(* Schneider Machine Expert - Basic project LT, file version 1.7.0.0 *)
(* ProjectInformations: Name=New project *)

HARDWARE
  Cpu 0: TM221ME32TK
  EthernetConfiguration: NetworkName=M221, IpAllocationMode=FixedAddress, IpAddress=0.0.0.0, SubnetMask=0.0.0.0
  SerialLineConfiguration: Baud=Baud19200, Parity=ParityEven, DataBits=DataBits8, StopBits=StopBits1, PhysicalMedium=PhysicalMediumRs485, TransmissionMode=TransmissionModeModbusRtu, SlaveId=1, Addressing=SlaveAddressing
  MastTask: UsePeriodScanMode=false, PeriodScan=100
  FastTask: Period=255
  CpuBehavior: StartingMode=StartAsPreviousState, AutoSaveRamOnEeprom=true, WatchdogPeriod=250

SYMBOLS  (address, symbol, comment, settings)
  %Q0.0       "P1"
  %Q0.1       "P2"
  %Q0.2       "SOV"
  %IW0.0      [Type=Type_0_10V, Scope=Scope_Normal, Minimum=0, Maximum=1000]

POU New POU
  (* SectionNumber=1 *)

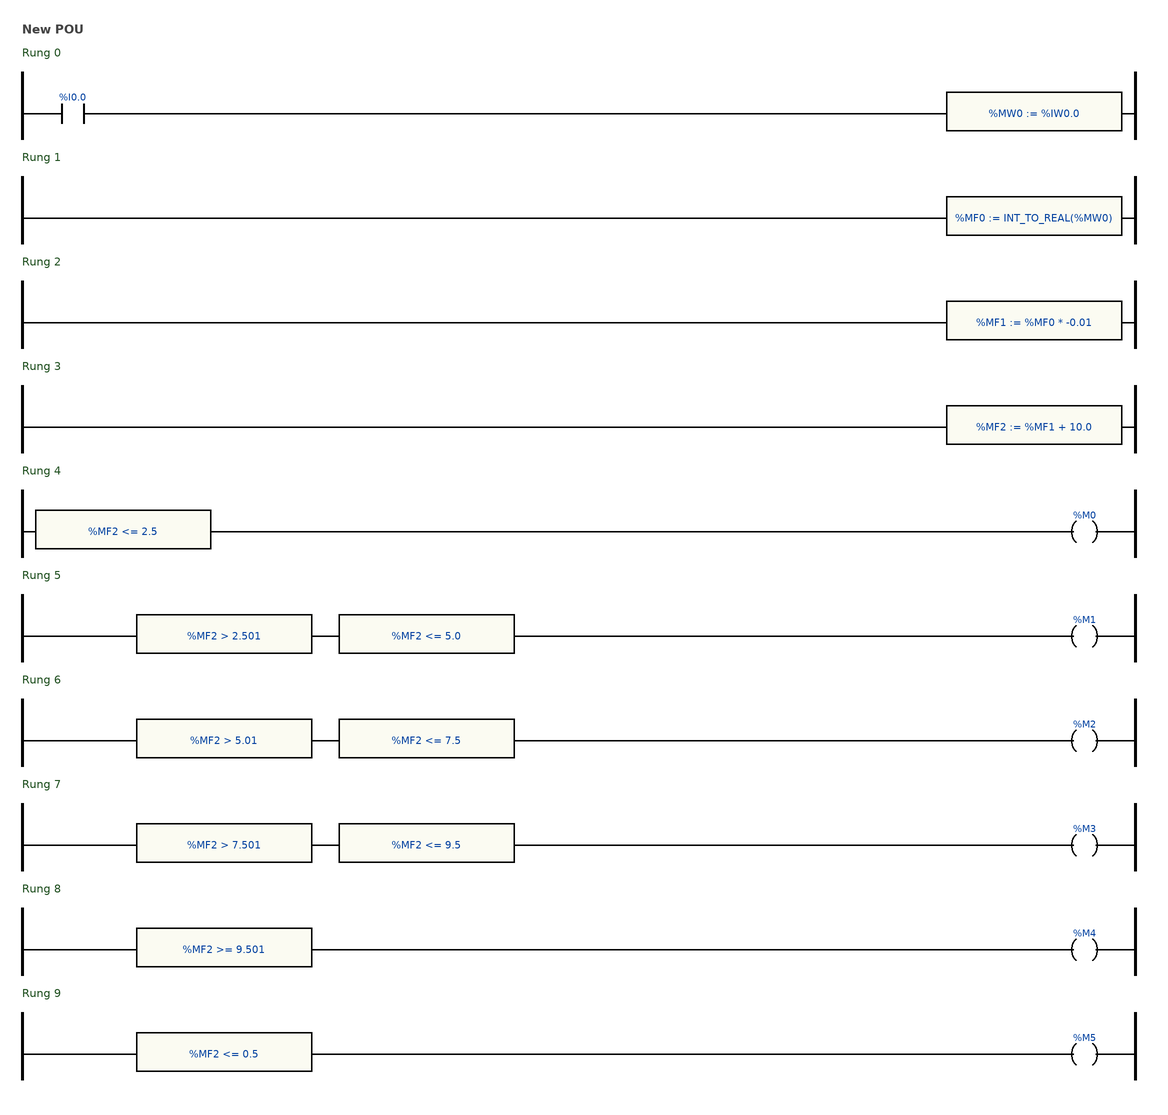

// Rung 0
  LD %I0.0
  [ %MW0 := %IW0.0 ]
  // as ST:
  //   IF %I0.0 THEN %MW0 := %IW0.0; END_IF;

// Rung 1
  LD 1
  [ %MF0 := INT_TO_REAL ( %MW0 ) ]
  // as ST:
  //   %MF0 := INT_TO_REAL ( %MW0 );

// Rung 2
  LD 1
  [ %MF1 := %MF0 * -0.01 ]
  // as ST:
  //   %MF1 := %MF0  *  -0.01;

// Rung 3
  LD 1
  [ %MF2 := %MF1 + 10.0 ]
  // as ST:
  //   %MF2 := %MF1  +  10.0;

// Rung 4
  LD [ %MF2 <= 2.5 ]
  ST %M0
  // as ST:
  //   %M0 := %MF2 <= 2.5;

// Rung 5
  LD [ %MF2 > 2.501 ]
  AND [ %MF2 <= 5.0 ]
  ST %M1
  // as ST:
  //   %M1 := %MF2 > 2.501 AND %MF2 <= 5.0;

// Rung 6
  LD [ %MF2 > 5.01 ]
  AND [ %MF2 <= 7.5 ]
  ST %M2
  // as ST:
  //   %M2 := %MF2 > 5.01 AND %MF2 <= 7.5;

// Rung 7
  LD [ %MF2 > 7.501 ]
  AND [ %MF2 <= 9.5 ]
  ST %M3
  // as ST:
  //   %M3 := %MF2 > 7.501 AND %MF2 <= 9.5;

// Rung 8
  LD [ %MF2 >= 9.501 ]
  ST %M4
  // as ST:
  //   %M4 := %MF2 >= 9.501;

// Rung 9
  LD [ %MF2 <= 0.5 ]
  ST %M5
  // as ST:
  //   %M5 := %MF2 <= 0.5;

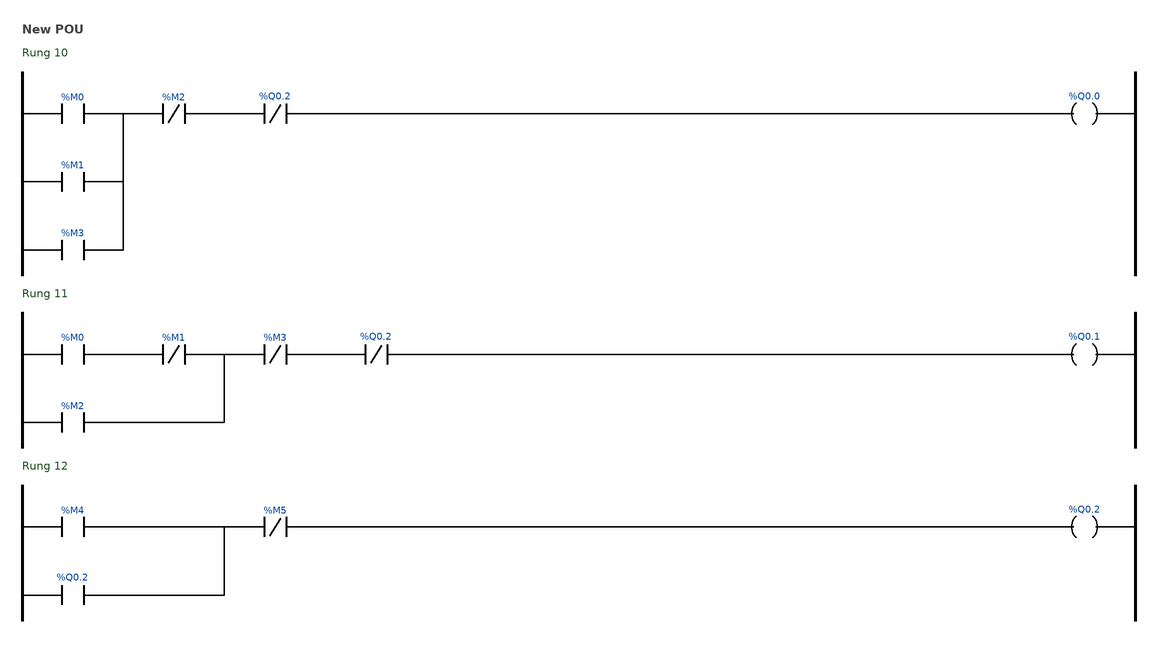

// Rung 10
  LD %M0
  OR %M1
  OR %M3
  ANDN %M2
  ANDN %Q0.2
  ST %Q0.0
  // as ST:
  //   %Q0.0 := (%M0 OR %M1 OR %M3) AND NOT %M2 AND NOT %Q0.2;

// Rung 11
  LD %M0
  ANDN %M1
  OR %M2
  ANDN %M3
  ANDN %Q0.2
  ST %Q0.1
  // as ST:
  //   %Q0.1 := (%M0 AND NOT %M1 OR %M2) AND NOT %M3 AND NOT %Q0.2;

// Rung 12
  LD %M4
  OR %Q0.2
  ANDN %M5
  ST %Q0.2
  // as ST:
  //   %Q0.2 := (%M4 OR %Q0.2) AND NOT %M5;
